// TIA Portal project "NastroConta3" (V17)
// Vorlageprojekt für das Buch mit Zielsystem S7-1200

(* hardware
DEVICE "S7-1200-Station_1"  S7-1200 Station
   slot 0: "Baugruppenträger_0"  Rack  V1.0
   slot 1: "PLC_1"  CPU 1211C DC/DC/DC  6ES7 211-1AE40-0XB0  V4.1
*)

// ===== PLC "PLC_1"  CPU 1211C DC/DC/DC =====

VAR_GLOBAL   // PLC tag table "Standard-Variablentabelle"
   "AVA1" AT %Q0.0 : Bool;   // Fa avanzare nastro iniziale
   "AVA2" AT %Q0.1 : Bool;   // Fa avanzare nastro contatore
   "I_READY" AT %I0.0 : Bool;   // Sensore nastro_iniziale
   "SI" AT %I0.1 : Bool;
   "SF" AT %I0.2 : Bool;
END_VAR

DATA_BLOCK "Sistema_DB"   // DB1
{ S7_Optimized_Access := 'TRUE' }
VERSION : 0.1
// stored: InstanceOfName Sistema
"Sistema"
BEGIN
END_DATA_BLOCK

FUNCTION_BLOCK "Nastro"   // FB1, LAD
{ S7_Optimized_Access := 'TRUE' }
VERSION : 0.1
   VAR_INPUT
      S : Bool;
      P_DOPO : Bool;
   END_VAR
   VAR_OUTPUT
      AVA : Bool;
      P_CONS : Bool;
      P_ACC : Bool;
   END_VAR
   VAR
      INIT : Bool;
      F0 : Bool;
      F1 : Bool;
      TR0 : Bool;
      TR1 : Bool;
   END_VAR
   VAR_TEMP   // added for the SCL form of the ladder/FBD networks
      _w1 : Bool;
   END_VAR
BEGIN

REGION Network 1: INIZIALIZZAZIONE
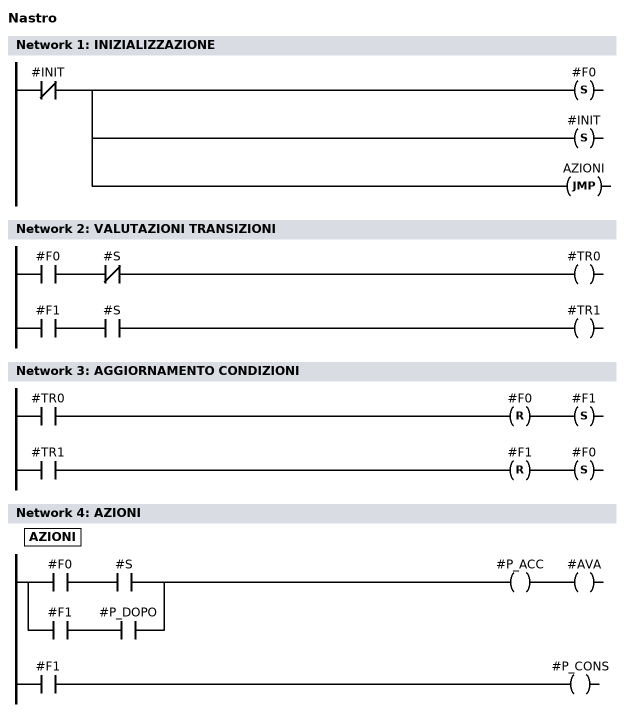
   RUNG wire#powerrail
      I_Contact( #INIT )
      wire#w1
      S_Coil( #F0 )
   END_RUNG
   RUNG wire#w1
      S_Coil( #INIT )
   END_RUNG
   RUNG wire#w1
      JumpCoil( AZIONI )
   END_RUNG
   // the same network as SCL:
   IF NOT #INIT THEN #F0 := TRUE; END_IF;
   #_w1 := NOT #INIT;
   IF #_w1 THEN
       #INIT := TRUE;
       GOTO AZIONI;
   END_IF;
END_REGION

REGION Network 2: VALUTAZIONI TRANSIZIONI
   RUNG wire#powerrail
      Contact( #F0 )
      I_Contact( #S )
      Coil( #TR0 )
   END_RUNG
   RUNG wire#powerrail
      Contact( #F1 )
      Contact( #S )
      Coil( #TR1 )
   END_RUNG
   // the same network as SCL:
   #TR0 := #F0 AND NOT #S;
   #TR1 := #F1 AND #S;
END_REGION

REGION Network 3: AGGIORNAMENTO CONDIZIONI
   RUNG wire#powerrail
      Contact( #TR0 )
      R_Coil( #F0 )
      S_Coil( #F1 )
   END_RUNG
   RUNG wire#powerrail
      Contact( #TR1 )
      R_Coil( #F1 )
      S_Coil( #F0 )
   END_RUNG
   // the same network as SCL:
   IF #TR0 THEN
       #F0 := FALSE;
       #F1 := TRUE;
   END_IF;
   IF #TR1 THEN
       #F1 := FALSE;
       #F0 := TRUE;
   END_IF;
END_REGION

REGION Network 4: AZIONI
   Label( AZIONI )
   RUNG wire#powerrail
      Contact( #F0 )
      Contact( #S )
      wire#w1
      Coil( #P_ACC )
      Coil( #AVA )
   END_RUNG
   RUNG wire#powerrail
      Contact( #F1 )
      Contact( #P_DOPO )
   END_RUNG wire#w1
   RUNG wire#powerrail
      Contact( #F1 )
      Coil( #P_CONS )
   END_RUNG
   // the same network as SCL:
   AZIONI:
   #P_ACC := (#F0 AND #S) OR (#F1 AND #P_DOPO);
   #AVA := #P_ACC;
   #P_CONS := #F1;
END_REGION
END_FUNCTION_BLOCK

FUNCTION_BLOCK "NastroContatore"   // FB2, LAD
{ S7_Optimized_Access := 'TRUE' }
VERSION : 0.1
   VAR_INPUT
      SI : Bool;
      SF : Bool;
      P_DOPO : Bool;
   END_VAR
   VAR_OUTPUT
      AVA : Bool;
      P_ACC : Bool;
      P_CONS : Bool;
   END_VAR
   VAR
      INIT : Bool;
      F0 : Bool;
      F1 : Bool;
      TR0 : Bool;
      TR1 : Bool;
      "MEMO-1" : Bool;
      "MEMO-2" : Bool;
      "MEMO-3" : Bool;
      "MEMO-4" : Bool;
      C1 : CTU_INT;
      C2 : CTU_INT;
   END_VAR
   VAR RETAIN
      RESET1 : Bool;
      RESET2 : Bool;
   END_VAR
   VAR_TEMP   // added for the SCL form of the ladder/FBD networks
      _w1 : Bool;
      _w2 : Bool;
      _w3 : Bool;
      _w4 : Bool;
   END_VAR
   // C1.PV := 3;
   // C2.PV := 3;
BEGIN

REGION Network 1: INIZIALIZZAZIONE
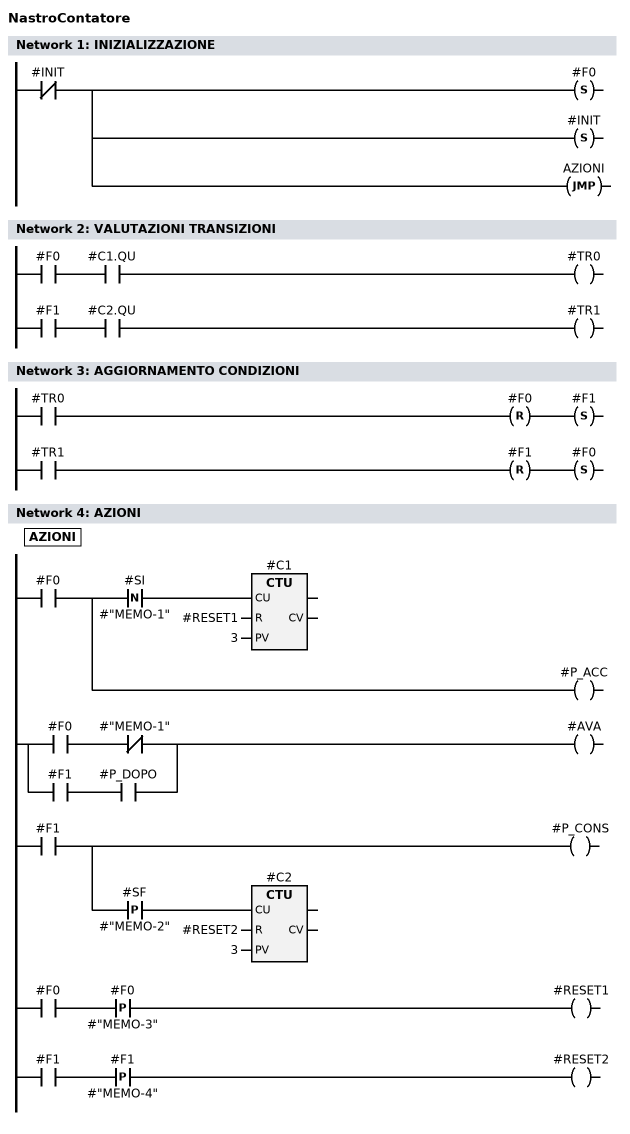
   RUNG wire#powerrail
      I_Contact( #INIT )
      wire#w1
      S_Coil( #F0 )
   END_RUNG
   RUNG wire#w1
      S_Coil( #INIT )
   END_RUNG
   RUNG wire#w1
      JumpCoil( AZIONI )
   END_RUNG
   // the same network as SCL:
   IF NOT #INIT THEN #F0 := TRUE; END_IF;
   #_w1 := NOT #INIT;
   IF #_w1 THEN
       #INIT := TRUE;
       GOTO AZIONI;
   END_IF;
END_REGION

REGION Network 2: VALUTAZIONI TRANSIZIONI
   RUNG wire#powerrail
      Contact( #F0 )
      Contact( #C1.QU )
      Coil( #TR0 )
   END_RUNG
   RUNG wire#powerrail
      Contact( #F1 )
      Contact( #C2.QU )
      Coil( #TR1 )
   END_RUNG
   // the same network as SCL:
   #TR0 := #F0 AND #C1.QU;
   #TR1 := #F1 AND #C2.QU;
END_REGION

REGION Network 3: AGGIORNAMENTO CONDIZIONI
   RUNG wire#powerrail
      Contact( #TR0 )
      R_Coil( #F0 )
      S_Coil( #F1 )
   END_RUNG
   RUNG wire#powerrail
      Contact( #TR1 )
      R_Coil( #F1 )
      S_Coil( #F0 )
   END_RUNG
   // the same network as SCL:
   IF #TR0 THEN
       #F0 := FALSE;
       #F1 := TRUE;
   END_IF;
   IF #TR1 THEN
       #F1 := FALSE;
       #F0 := TRUE;
   END_IF;
END_REGION

REGION Network 4: AZIONI
   AZIONI:
   #_w1 := #F0 AND NOT #SI AND #"MEMO-1";   // falling edge of #SI
   #"MEMO-1" := #SI;
   #C1(CU := #_w1, R := #RESET1, PV := 3);   // CTU
   #P_ACC := #F0;
   #AVA := (#F0 AND NOT #"MEMO-1") OR (#F1 AND #P_DOPO);
   #P_CONS := #F1;
   #_w2 := #F1 AND #SF AND NOT #"MEMO-2";   // rising edge of #SF
   #"MEMO-2" := #SF;
   #C2(CU := #_w2, R := #RESET2, PV := 3);   // CTU
   #_w3 := #F0 AND #F0 AND NOT #"MEMO-3";   // rising edge of #F0
   #"MEMO-3" := #F0;
   #RESET1 := #_w3;
   #_w4 := #F1 AND #F1 AND NOT #"MEMO-4";   // rising edge of #F1
   #"MEMO-4" := #F1;
   #RESET2 := #_w4;
END_REGION
END_FUNCTION_BLOCK

FUNCTION_BLOCK "Sistema"   // FB3, FBD
{ S7_Optimized_Access := 'TRUE' }
VERSION : 0.1
   VAR
      Nastro_iniziale : "Nastro";
      Nastro_contatore : "NastroContatore";
   END_VAR
BEGIN

REGION Network 1
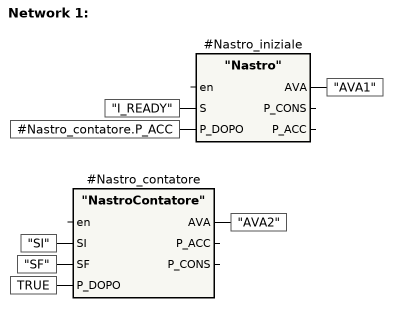
   #Nastro_iniziale(S := "I_READY", P_DOPO := #Nastro_contatore.P_ACC, AVA => "AVA1");   // "Nastro"
   #Nastro_contatore(SI := "SI", SF := "SF", P_DOPO := TRUE, AVA => "AVA2");   // "NastroContatore"
END_REGION
END_FUNCTION_BLOCK

FUNCTION "MHJ-PLC-Lab-Function-S71200" : Void   // FC9000, SCL
{ S7_Optimized_Access := 'TRUE' }
VERSION : 0.1
   VAR_TEMP
      rdTimeReturn : Int;
      outputTime : DTL;
      SyncVal : Byte;
      forVal : Int;
      forVal_2 : Int;
      Value : Byte;
   END_VAR
   VAR CONSTANT
      CompVal : Byte := 16#34;
      Value_01 : Byte := 16#11;
      Value_01_DW : DWord := 16#A165_D992;
      Value_02_DW : DWord := 16#58BE_4401;
   END_VAR
BEGIN

   #Value:=PEEK(area := 16#82,
        dbNumber := 0,
        byteOffset := 511);
   #Value := #Value + 1;

   POKE(area := 16#82,
        dbNumber := 0,
        byteOffset := 511,
        value := #Value);

   POKE(area:=16#81,
        dbNumber:=0,
        byteOffset:=1016,
        value:=#Value_01_DW);
   POKE(area := 16#81,
        dbNumber := 0,
        byteOffset := 1020,
        value := #Value_02_DW);

   POKE(area := 16#81,
        dbNumber := 0,
        byteOffset := 511,
        value := B#16#00);

   FOR #forVal := 0 TO 120 DO
       FOR #forVal_2:=0 TO 10 DO
           #rdTimeReturn:=RD_SYS_T(#outputTime);
           #rdTimeReturn := WR_SYS_T(#outputTime);
           #rdTimeReturn := RD_SYS_T(#outputTime);
           #rdTimeReturn := WR_SYS_T(#outputTime);
       END_FOR;
       #SyncVal:= PEEK(area := 16#81,
                      dbNumber := 0,
                      byteOffset := 511);
       IF #SyncVal = #CompVal THEN
          GOTO M_1;
       END_IF;
   END_FOR;
   RETURN;

   M_1:
   POKE(area := 16#81,
        dbNumber := 0,
        byteOffset := 511,
        value := B#16#0);
END_FUNCTION

ORGANIZATION_BLOCK "Main"   // OB1, FBD, ProgramCycle
TITLE = "Main Program Sweep (Cycle)"
{ S7_Optimized_Access := 'TRUE' }
VERSION : 0.1
   VAR_INPUT
      Initial_Call : Bool;   // Initial call of this OB
      Remanence : Bool;   // =True, if remanent data are available
   END_VAR
BEGIN

REGION Network 1: Konnektierungsbaustein für PLC-Lab
   // Im Netzwerk 1 wird der Konnektierungsbaustein für PLC-Lab aufgerufen.
   // Dieser Aufruf darf nicht entfernt werden!
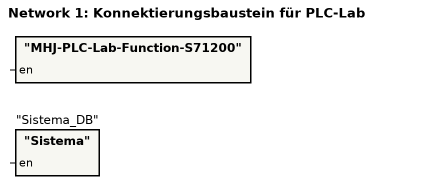
   "MHJ-PLC-Lab-Function-S71200"();
   "Sistema_DB"();   // "Sistema"
END_REGION

REGION Network 2: Ihr Programm
   // Schreiben Sie ab Netzwerk 2 Ihr Programm
END_REGION
END_ORGANIZATION_BLOCK